KUKA KRL program: R2_MillingInit.src

&ACCESS RV1
DEF R2_MillingInit ( )

   ;******************************************************
   ;*             Reset signals on startup               *
   ;******************************************************
   gbRobControlActive   = FALSE
   gDOSpindleEnable     = FALSE
   gbSpindleStart      = FALSE

   oFreqconverterCtlw = gsSpindleWord.WaitForCommand
   oConverterSetSpeed = 0

END
